TYPE EL2819_Data :
STRUCT
	{attribute addProperty Name "DIG Diag Inputs"}
	_diag : EL2819_Diag;
	{attribute addProperty Name "DIG Inputs Device"}
	_inputs : stDIGInputsDevice;
	{attribute addProperty Name "DIG Outputs"}
	_outputs : EL2819_Outputs;
END_STRUCT
END_TYPE

(* stored: Version 1.1.0.1, ProductVersion 3.1.4024.9
   DUT EL2819_Data: Id {8f7c03d0-5afb-0ebd-0e01-3ba2f298e76f} *)
